// TIA Portal V19 export
TYPE "C402_STU_IF_M33_TYPIC"
   STRUCT
      CMD_AAN { ExternalAccessible := 'False'; ExternalVisible := 'False'; ExternalWritable := 'False'} : Bool;   // TRUE = weergeven beeldstand verkeerslicht FALSE = niets weergeven
      CMD_RES { ExternalAccessible := 'False'; ExternalVisible := 'False'; ExternalWritable := 'False'} : Bool;   // Reset van de latched storingen
   END_STRUCT;
END_TYPE
